Omron CX-Programmer project NewProject (CX-Programmer 9.61)

# PLC NewPLC1: CP1H XA
; 2022.06.30 / lecture works

## Global symbols (name address type ; comment)
0.00 BOOL  ; Start
0.01 BOOL  ; Stop
10.00 BOOL  ; Conv

## Program NewProgram1 (cyclic task 0)

### Section Section1

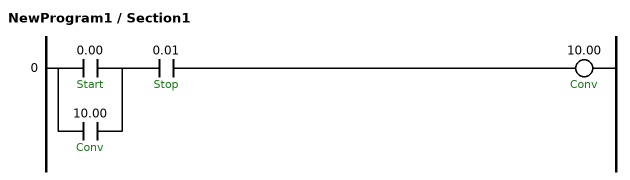
; rung 0
LD 0.00  ; Start
OR 10.00  ; Conv
AND 0.01  ; Stop
OUT 10.00  ; Conv

### Section END
; rung 0
END(001)